PROGRAM ConvertIO
VAR
	wRealPower AT %I*: WORD := 0;
	iTemperatureSensor AT %I*: INT := 0;
	byHeaterActuator AT %Q*: BYTE := 0;
END_VAR

GVL.rTempSensor := INT_TO_REAL(iTemperatureSensor) / 10;
byHeaterActuator := REAL_TO_BYTE((GVL.iHeaterActuator * 50) / 100);
GVL.iRealPower := WORD_TO_INT(wRealPower);

END_PROGRAM

(* stored: Version 1.1.0.1, ProductVersion 3.1.4024.12
   POU ConvertIO: Id {0580372f-3c7b-44c1-bbdf-2b88f1dab63c}, SpecialFunc None *)
